TYPE ST_ProcessResult :
STRUCT
	bValid          : BOOL;
    bPassed         : BOOL;
    eCode           : E_ProcessResultCode;
    udiFaultCode    : UDINT;
    udiAlertCode    : UDINT;
    usiRecipe       : USINT;
    lrDispenseValue : LREAL;
    sDetail         : STRING(120);
END_STRUCT
END_TYPE

(* stored: Version 1.1.0.1, ProductVersion 3.1.4026.18
   DUT ST_ProcessResult: Id {c3de95b9-d31b-45c1-a11a-e047ded3904c} *)
